FUNCTION_BLOCK COLOR_PURPLE (* constant *)
  (* Standard: ISO 11783-6 *)
  (* Version 1.0, 2022-07-29, franz *)
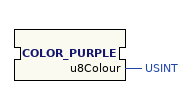
  VAR_OUTPUT
    u8Colour : USINT; (* Colour *)
  END_VAR
END_FUNCTION_BLOCK
